Yaskawa INFORM job: muffler_cylinder_program.JBI

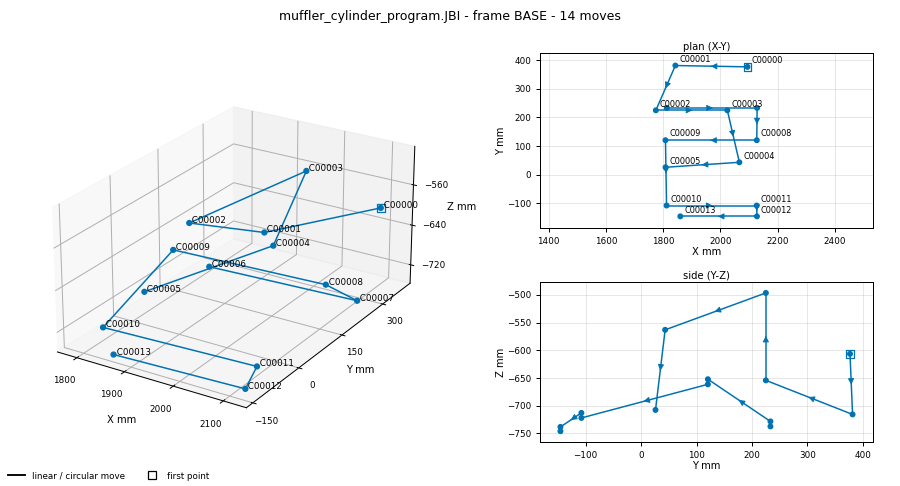
[picture p0: tool path of muffler_cylinder_program.JBI in frame BASE, 14 of 19 moves have a stored position in this frame; points joined in program order, loops and branches not executed]
/JOB
//NAME muffler_cylinder_program
//POS
///NPOS 14,0,14,0,0,0
///TOOL 0
///POSTYPE BASE
///RECTAN
///RCONF 0,0,0,0,0,0,0,0,0,0,0,0,0,0,0,0,0,0,0,0,0,0,0,0
C00000=2094.997421,376.855033,-606.366987,175.000000,-75.636078,-80.694767
C00001=1843.045643,381.482414,-715.581805,175.000000,-60.000000,-80.694767
C00002=1774.902201,225.039714,-654.116740,175.000000,-33.237144,-15.522161
C00003=2024.644346,225.039697,-496.427820,175.000000,-33.237144,-15.522161
C00004=2066.646085,43.346405,-562.988155,175.000000,-61.207273,69.695178
C00005=1808.613070,25.953977,-707.492503,175.000000,-60.000000,69.695178
C00006=1813.202155,233.328367,-737.255431,175.000000,-60.000000,-89.487041
C00007=2128.736245,233.328375,-728.173156,175.000000,-60.000000,-89.487041
C00008=2127.489377,120.483464,-652.096718,156.550702,-5.000000,5.000000
C00009=1808.440137,120.483455,-661.280173,156.550702,-5.000000,5.000000
C00010=1812.259611,-107.761220,-721.940798,175.000000,-53.257721,88.768743
C00011=2127.296847,-107.761212,-712.872824,175.000000,-53.257721,88.768743
C00012=2127.988371,-145.566954,-738.160812,175.000000,-60.000000,89.915372
C00013=1860.308839,-145.566962,-745.865651,175.000000,-60.000000,89.915372
///POSTYPE PULSE
///PULSE
EX00000=349184.0
EX00001=363520.0
///POSTYPE PULSE
///PULSE
EC00000=349184.0
EC00001=349184.0
EC00002=349184.0
EC00003=349184.0
EC00004=349184.0
EC00005=349184.0
EC00006=363520.0
EC00007=363520.0
EC00008=363520.0
EC00009=363520.0
EC00010=363520.0
EC00011=363520.0
EC00012=363520.0
EC00013=363520.0
//INST
///DATE 2023/08/15 14:43
///ATTR SC,RW,RJ
////FRAME BASE
///GROUP1 RB1,ST1
NOP
MOVJ P009 EX000 VJ=15.00
MOVJ C00000 EC00000 VJ=15.0
CALL JOB:SPYON
MOVL C00001 EC00001 V=150.0
MOVL C00002 EC00002 V=150.0
MOVL C00003 EC00003 V=150.0
MOVL C00004 EC00004 V=150.0
MOVL C00005 EC00005 V=150.0
CALL JOB:SPYOF
MOVJ P009 VJ=15.00
MOVL P009 EX00000 V=150.0
MOVJ C00006 EC00006 VJ=15.0
CALL JOB:SPYON
MOVL C00007 EC00007 V=150.0
MOVL C00008 EC00008 V=150.0
MOVL C00009 EC00009 V=150.0
MOVL C00010 EC00010 V=150.0
MOVL C00011 EC00011 V=150.0
MOVL C00012 EC00012 V=150.0
MOVL C00013 EC00013 V=150.0
CALL JOB:SPYOF
MOVJ P009 VJ=15.00
MOVL P009 EX00001 V=150.0
END
